# EPICS autosave request: scripts/spixconv/server/autosave/spixconv.req
$(P):IPAddress.VAL
$(P):BoardAddress.VAL
